PROGRAM P_Section_3
VAR
END_VAR

P_Example_Stopwatch();

END_PROGRAM

(* stored: Version 1.1.0.1, ProductVersion 3.1.4024.4
   POU P_Section_3: Id {9dfa112c-c28e-495f-b48c-fe41abc3434c}, SpecialFunc None *)
